// TIA Portal V20 export
// export: Created 2026-09-14T11:29:00.8575237Z, ExportSetting None, DisplayName Totally Integrated Automation Portal, DisplayVersion V20, DisplayName TIA Portal Openness, DisplayVersion V20, DisplayName TIA Portal Version Control Interface, DisplayVersion V20, DisplayName STEP 7 Professional, DisplayVersion V20, DisplayName STEP 7 Safety, DisplayVersion V20, DisplayName WinCC Basic/Comfort/Advanced, DisplayVersion V20, DisplayName WinCC Unified, DisplayVersion V20
TYPE "LMQTT_typePublishData"
   STRUCT
      publishMessage : Bool;   // Set to true. Can be reset to false once done flag is set be FB
      publishTopic : WString[250];   // Size be increased, but must increase MAX_SENDBUFFER and MAX_PUBLISH_MESSAGE in the FB
      publishMessageData : WString[800];   // Size be increased, but must increase MAX_SENDBUFFER and MAX_PUBLISH_MESSAGE in the FB
      publishQoS : Int;   // Defines the QoS level for the MQTT message. 0,1 and 2 supported
      publishRetainFlag : Bool;   // If true, message may be saved at the broker
   END_STRUCT;
END_TYPE
